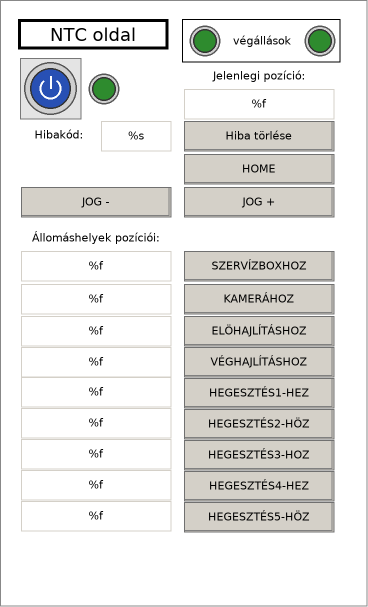
VISUALIZATION Tengely_NTC  // 368x607
    PowerSwitch (20,58 61x61), variable: GVL.bJozsiServo, behaviour: TOGGLE, style: Switch-PowerSwitch-Blue
    Button (184,154 150x30), "HOME"
        OnMouseUp: execute { JOZSITENGELY.sJozsiAxisCommand:='HOME'; }
    Button (184,187 150x30), "JOG +"
        tap JOZSITENGELY.bJozsiJOGPlus
    Button (21,187 150x30), "JOG -"
        tap JOZSITENGELY.bJozsiJOGMinus
    Button (184,121 150x30), "Hiba törlése"
        tap JOZSITENGELY.bJozsiReset
    Textfield (101,121 70x30), "%s", text variable: JOZSITENGELY.nJozsiErrorCode, input disabled if: TRUE
    Textfield (21,316 150x30), "%f", text variable: GVL.lrHajlitoPosition1
    Button (184,316 150x30), "ELÖHAJLÍTÁSHOZ"
        OnMouseUp: execute { JOZSITENGELY.lrJozsiPosition:=GVL.lrHajlitoPosition1; JOZSITENGELY.sJozsiAxisCommand:='MOVE'; }
    Textfield (184,89 150x30), "%f", text variable: JOZSITENGELY.lrJozsiActPos, input disabled if: TRUE
    Label (184,66 150x20), "Jelenlegi pozíció:"
    Textfield (21,284 150x30), "%f", text variable: GVL.lrNTCKameraPosition
    Button (184,284 150x30), "KAMERÁHOZ"
        OnMouseUp: execute { JOZSITENGELY.lrJozsiPosition:=GVL.lrNTCKameraPosition; JOZSITENGELY.sJozsiAxisCommand:='MOVE'; }
    Textfield (21,377 150x30), "%f", text variable: GVL.lrHegesztoPosition1
    Button (184,378 150x30), "HEGESZTÉS1-HEZ"
        OnMouseUp: execute { JOZSITENGELY.lrJozsiPosition:=GVL.lrHegesztoPosition1; JOZSITENGELY.sJozsiAxisCommand:='MOVE'; }
    Textfield (21,408 150x30), "%f", text variable: GVL.lrHegesztoPosition2
    Button (184,409 150x30), "HEGESZTÉS2-HÖZ"
        OnMouseUp: execute { JOZSITENGELY.lrJozsiPosition:=GVL.lrHegesztoPosition2; JOZSITENGELY.sJozsiAxisCommand:='MOVE'; }
    Textfield (21,439 150x30), "%f", text variable: GVL.lrHegesztoPosition3
    Button (184,440 150x30), "HEGESZTÉS3-HOZ"
        OnMouseUp: execute { JOZSITENGELY.lrJozsiPosition:=GVL.lrHegesztoPosition3; JOZSITENGELY.sJozsiAxisCommand:='MOVE'; }
    Textfield (21,470 150x30), "%f", text variable: GVL.lrHegesztoPosition4
    Button (184,471 150x30), "HEGESZTÉS4-HEZ"
        OnMouseUp: execute { JOZSITENGELY.lrJozsiPosition:=GVL.lrHegesztoPosition4; JOZSITENGELY.sJozsiAxisCommand:='MOVE'; }
    Textfield (21,501 150x30), "%f", text variable: GVL.lrHegesztoPosition5
    Button (184,502 150x30), "HEGESZTÉS5-HÖZ"
        OnMouseUp: execute { JOZSITENGELY.lrJozsiPosition:=GVL.lrHegesztoPosition5; JOZSITENGELY.sJozsiAxisCommand:='MOVE'; }
    Label (297,575 69x30)
    Button (184,251 150x30), "SZERVÍZBOXHOZ"
        OnMouseUp: execute { JOZSITENGELY.lrJozsiPosition:=GVL.lrNTCSzervizbox; JOZSITENGELY.sJozsiAxisCommand:='MOVE'; }
    Lamp1 (86,71 36x36), variable: JOZSITENGELY.bHomeReady, style: Lamp-Lamp1-Green
    Label (24,125 70x20), "Hibakód:"
    Label (21,228 150x20), "Állomáshelyek pozíciói:"
    RoundedRectangle (18,19 150x30)
    Label (18,20 150x30), "NTC oldal"
    Group (182,19 158x43)
        Rectangle (0,0 158x43)
        Lamp1 (5,4 36x36), variable: GVL.bJozsiNegSwitch, style: Lamp-Lamp1-Green
        Lamp1 (120,4 36x36), variable: GVL.bJozsiPosSwitch, style: Lamp-Lamp1-Green
        Label (45,12 70x20), "végállások"
    Textfield (21,251 150x30), "%f", text variable: GVL.lrNTCSzervizbox
    Textfield (21,347 150x30), "%f", text variable: GVL.lrHajlitoPosition2
    Button (184,347 150x30), "VÉGHAJLÍTÁSHOZ"
        OnMouseUp: execute { JOZSITENGELY.lrJozsiPosition:=GVL.lrHajlitoPosition2; JOZSITENGELY.sJozsiAxisCommand:='MOVE'; }
END_VISUALIZATION

(* stored: Version 1.1.0.1, ProductVersion 3.1.4024.11
   Visu Tengely_NTC: Id {98a2b511-3cbf-4056-9a9c-d5f71925da7d} *)
